// SIMATIC S7-200 project (STEP 7-Micro/WIN), CPU 221 REL 01.10

SYMBOL_TABLE USUARIO1
INICIAR          I0.0     // Switch para iniciar proceso (NA)
T1_MAX           I0.1     // Sensor capacitivo que detecta nivel máximo de tanque de mezclado.
T1_MED           I0.2     // Sensor capacitivo que detecta nivel medio de tanque de mezclado.
T1_MIN           I0.3     // Sensor capacitivo que detecta nivel mínimo de tanque de mezclado.
T2_MAX           I0.4     // Sensor capacitivo que detecta nivel máximo de tanque de llenado.
T2_MED           I0.5     // Sensor capacitivo que detecta nivel medio de tanque de llenado.
T2_MIN           I0.6     // Sensor capacitivo que detecta nivel mínimo de tanque de llenado.
S1               I0.7     // Sensor fotoeléctrico que detecta botella en posición para su llenado.
EV1              Q0.0     // Electroválvula que controla el flujo de agua
EV2              Q0.1     // Electroválvula que controla el flujo de cebada
EV3              Q0.2     // Electroválvula que controla el flujo de cerveza
MEZCLAR          Q0.3     // Motor que sirve para hacer la mezcla
EV4              Q0.4     // Electroválvula que controla el llenado de las botellas
BOTELLAS         Q0.5     // Activar despachador de botellas
END_SYMBOL_TABLE

ORGANIZATION_BLOCK PRINCIPAL:OB1
TITLE=
BEGIN
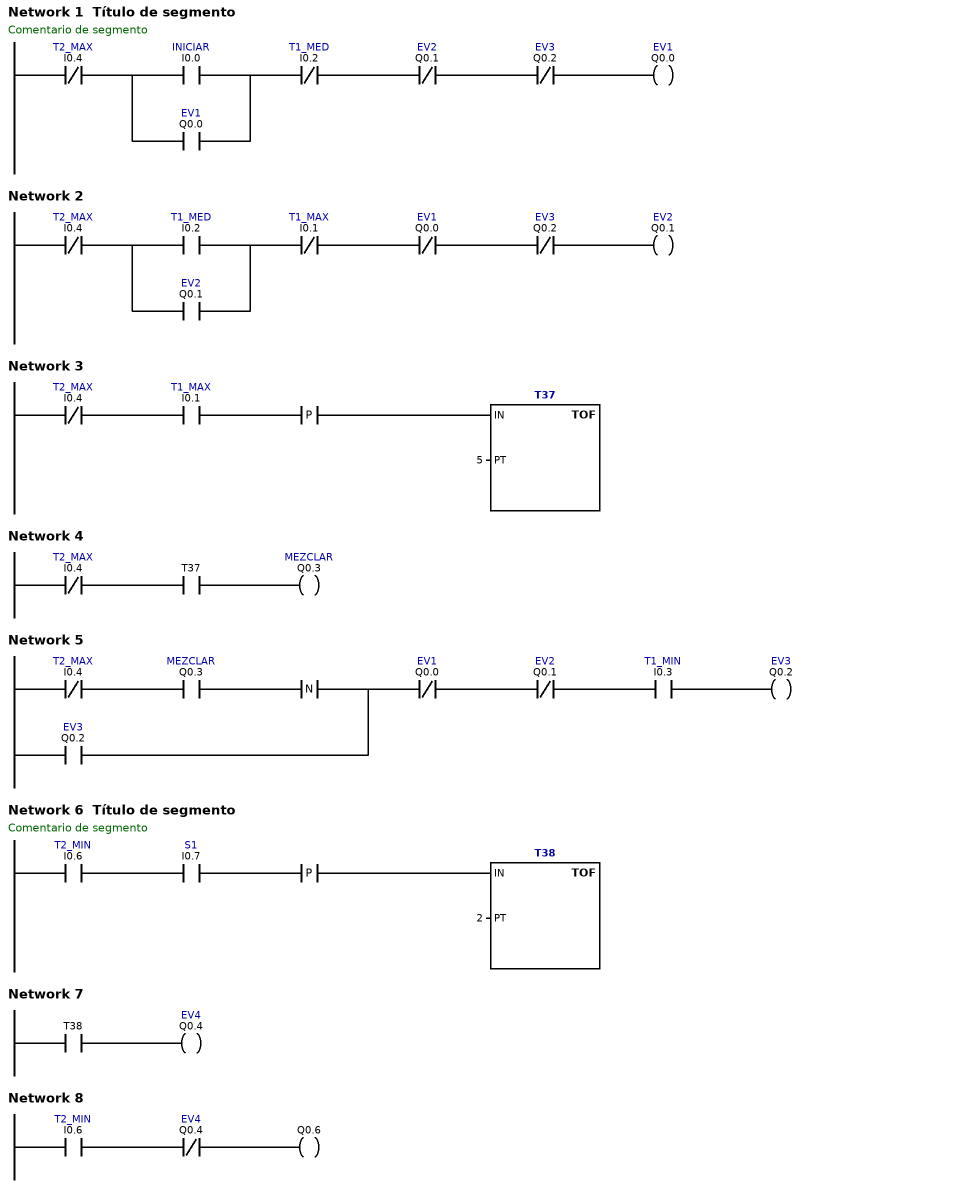
Network 1 // Título de segmento
// Comentario de segmento
LDN    T2_MAX:I0.4
LD     INICIAR:I0.0
O      EV1:Q0.0
ALD
AN     T1_MED:I0.2
AN     EV2:Q0.1
AN     EV3:Q0.2
=      EV1:Q0.0
Network 2
LDN    T2_MAX:I0.4
LD     T1_MED:I0.2
O      EV2:Q0.1
ALD
AN     T1_MAX:I0.1
AN     EV1:Q0.0
AN     EV3:Q0.2
=      EV2:Q0.1
Network 3
LDN    T2_MAX:I0.4
A      T1_MAX:I0.1
EU
TOF    T37, 5
Network 4
LDN    T2_MAX:I0.4
A      T37
=      MEZCLAR:Q0.3
Network 5
LDN    T2_MAX:I0.4
A      MEZCLAR:Q0.3
ED
O      EV3:Q0.2
AN     EV1:Q0.0
AN     EV2:Q0.1
A      T1_MIN:I0.3
=      EV3:Q0.2
Network 6 // Título de segmento
// Comentario de segmento
LD     T2_MIN:I0.6
A      S1:I0.7
EU
TOF    T38, 2
Network 7
LD     T38
=      EV4:Q0.4
Network 8
LD     T2_MIN:I0.6
AN     EV4:Q0.4
=      Q0.6
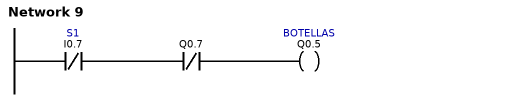
Network 9
LDN    S1:I0.7
AN     Q0.7
=      BOTELLAS:Q0.5
END_ORGANIZATION_BLOCK
